FUNCTION_BLOCK SPLIT_AD_INTO_AQ (* this Function splits the 16 AQ (QUARTER) adapters from a AD (DWORD) *)
  (* Standard: 61499-2; Description: Copyright (c) 2026 Meisterschulen am Ostbahnhof SPDX-License-Identifier: EPL-2.0 *)
  (* Version 1.0, 2026-05-16, Franz Höpfinger, Meisterschulen am Ostbahnhof, initial API and implementation and/or initial documentation *)
  PACKAGE adapter::splitting;
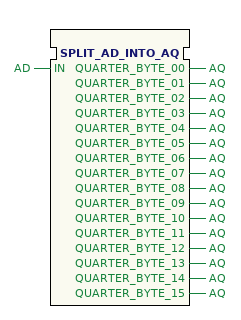
  SOCKETS
    IN : adapter::types::unidirectional::AD; (* DWORD Input *)
  END_SOCKETS
  PLUGS
    QUARTER_BYTE_00 : adapter::types::unidirectional::AQ; (* Quarter 0 *)
    QUARTER_BYTE_01 : adapter::types::unidirectional::AQ; (* Quarter 1 *)
    QUARTER_BYTE_02 : adapter::types::unidirectional::AQ; (* Quarter 2 *)
    QUARTER_BYTE_03 : adapter::types::unidirectional::AQ; (* Quarter 3 *)
    QUARTER_BYTE_04 : adapter::types::unidirectional::AQ; (* Quarter 4 *)
    QUARTER_BYTE_05 : adapter::types::unidirectional::AQ; (* Quarter 5 *)
    QUARTER_BYTE_06 : adapter::types::unidirectional::AQ; (* Quarter 6 *)
    QUARTER_BYTE_07 : adapter::types::unidirectional::AQ; (* Quarter 7 *)
    QUARTER_BYTE_08 : adapter::types::unidirectional::AQ; (* Quarter 8 *)
    QUARTER_BYTE_09 : adapter::types::unidirectional::AQ; (* Quarter 9 *)
    QUARTER_BYTE_10 : adapter::types::unidirectional::AQ; (* Quarter 10 *)
    QUARTER_BYTE_11 : adapter::types::unidirectional::AQ; (* Quarter 11 *)
    QUARTER_BYTE_12 : adapter::types::unidirectional::AQ; (* Quarter 12 *)
    QUARTER_BYTE_13 : adapter::types::unidirectional::AQ; (* Quarter 13 *)
    QUARTER_BYTE_14 : adapter::types::unidirectional::AQ; (* Quarter 14 *)
    QUARTER_BYTE_15 : adapter::types::unidirectional::AQ; (* Quarter 15 *)
  END_PLUGS
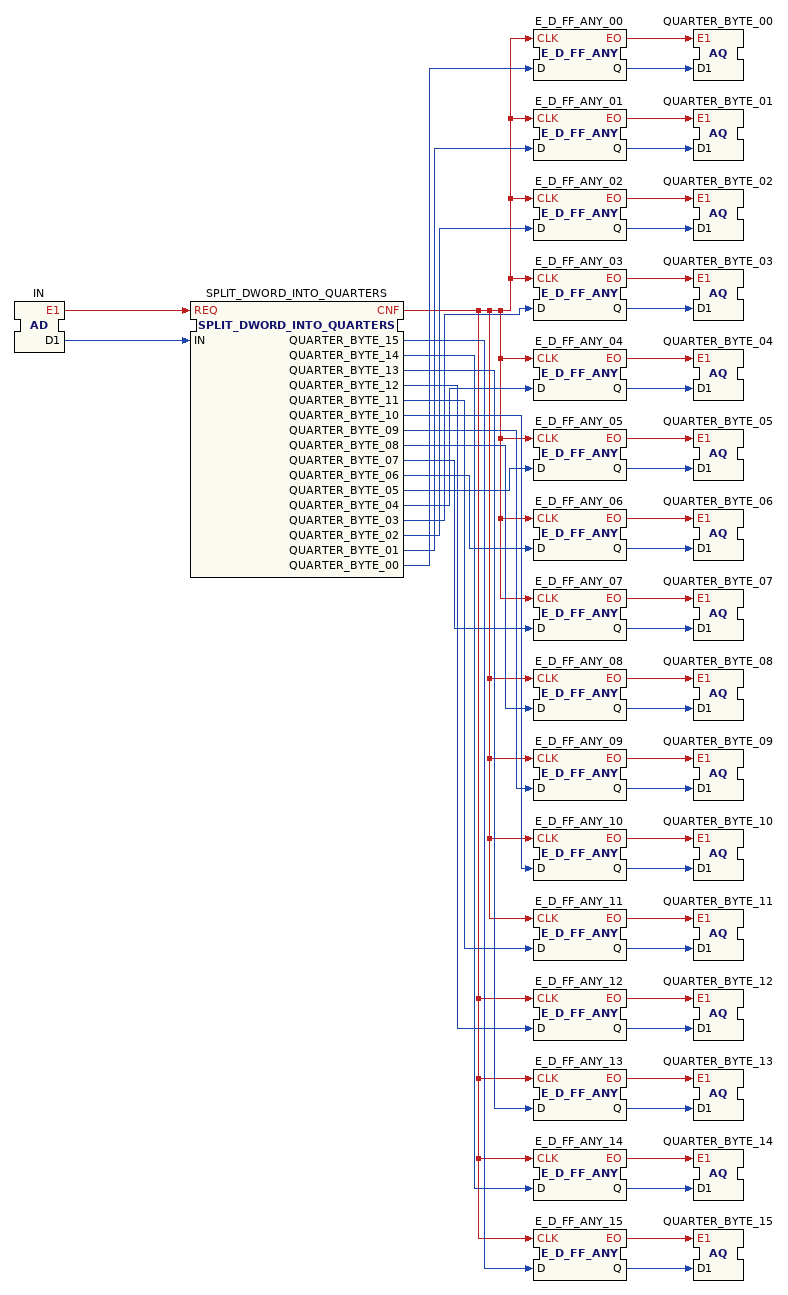
  FBS
    E_D_FF_ANY_00 : iec61499::events::E_D_FF_ANY;
    E_D_FF_ANY_01 : iec61499::events::E_D_FF_ANY;
    E_D_FF_ANY_02 : iec61499::events::E_D_FF_ANY;
    E_D_FF_ANY_03 : iec61499::events::E_D_FF_ANY;
    E_D_FF_ANY_04 : iec61499::events::E_D_FF_ANY;
    E_D_FF_ANY_05 : iec61499::events::E_D_FF_ANY;
    E_D_FF_ANY_06 : iec61499::events::E_D_FF_ANY;
    E_D_FF_ANY_07 : iec61499::events::E_D_FF_ANY;
    E_D_FF_ANY_08 : iec61499::events::E_D_FF_ANY;
    E_D_FF_ANY_09 : iec61499::events::E_D_FF_ANY;
    E_D_FF_ANY_10 : iec61499::events::E_D_FF_ANY;
    E_D_FF_ANY_11 : iec61499::events::E_D_FF_ANY;
    E_D_FF_ANY_12 : iec61499::events::E_D_FF_ANY;
    E_D_FF_ANY_13 : iec61499::events::E_D_FF_ANY;
    E_D_FF_ANY_14 : iec61499::events::E_D_FF_ANY;
    E_D_FF_ANY_15 : iec61499::events::E_D_FF_ANY;
    SPLIT_DWORD_INTO_QUARTERS : eclipse4diac::utils::splitting::SPLIT_DWORD_INTO_QUARTERS;
  END_FBS
  EVENT_CONNECTIONS
    IN.E1 TO SPLIT_DWORD_INTO_QUARTERS.REQ;
    SPLIT_DWORD_INTO_QUARTERS.CNF TO E_D_FF_ANY_00.CLK;
    SPLIT_DWORD_INTO_QUARTERS.CNF TO E_D_FF_ANY_01.CLK;
    SPLIT_DWORD_INTO_QUARTERS.CNF TO E_D_FF_ANY_02.CLK;
    SPLIT_DWORD_INTO_QUARTERS.CNF TO E_D_FF_ANY_03.CLK;
    SPLIT_DWORD_INTO_QUARTERS.CNF TO E_D_FF_ANY_04.CLK;
    SPLIT_DWORD_INTO_QUARTERS.CNF TO E_D_FF_ANY_05.CLK;
    SPLIT_DWORD_INTO_QUARTERS.CNF TO E_D_FF_ANY_06.CLK;
    SPLIT_DWORD_INTO_QUARTERS.CNF TO E_D_FF_ANY_07.CLK;
    SPLIT_DWORD_INTO_QUARTERS.CNF TO E_D_FF_ANY_08.CLK;
    SPLIT_DWORD_INTO_QUARTERS.CNF TO E_D_FF_ANY_09.CLK;
    SPLIT_DWORD_INTO_QUARTERS.CNF TO E_D_FF_ANY_10.CLK;
    SPLIT_DWORD_INTO_QUARTERS.CNF TO E_D_FF_ANY_11.CLK;
    SPLIT_DWORD_INTO_QUARTERS.CNF TO E_D_FF_ANY_12.CLK;
    SPLIT_DWORD_INTO_QUARTERS.CNF TO E_D_FF_ANY_13.CLK;
    SPLIT_DWORD_INTO_QUARTERS.CNF TO E_D_FF_ANY_14.CLK;
    SPLIT_DWORD_INTO_QUARTERS.CNF TO E_D_FF_ANY_15.CLK;
    E_D_FF_ANY_00.EO TO QUARTER_BYTE_00.E1;
    E_D_FF_ANY_01.EO TO QUARTER_BYTE_01.E1;
    E_D_FF_ANY_02.EO TO QUARTER_BYTE_02.E1;
    E_D_FF_ANY_03.EO TO QUARTER_BYTE_03.E1;
    E_D_FF_ANY_04.EO TO QUARTER_BYTE_04.E1;
    E_D_FF_ANY_05.EO TO QUARTER_BYTE_05.E1;
    E_D_FF_ANY_06.EO TO QUARTER_BYTE_06.E1;
    E_D_FF_ANY_07.EO TO QUARTER_BYTE_07.E1;
    E_D_FF_ANY_08.EO TO QUARTER_BYTE_08.E1;
    E_D_FF_ANY_09.EO TO QUARTER_BYTE_09.E1;
    E_D_FF_ANY_10.EO TO QUARTER_BYTE_10.E1;
    E_D_FF_ANY_11.EO TO QUARTER_BYTE_11.E1;
    E_D_FF_ANY_12.EO TO QUARTER_BYTE_12.E1;
    E_D_FF_ANY_13.EO TO QUARTER_BYTE_13.E1;
    E_D_FF_ANY_14.EO TO QUARTER_BYTE_14.E1;
    E_D_FF_ANY_15.EO TO QUARTER_BYTE_15.E1;
  END_CONNECTIONS
  DATA_CONNECTIONS
    IN.D1 TO SPLIT_DWORD_INTO_QUARTERS.IN;
    SPLIT_DWORD_INTO_QUARTERS.QUARTER_BYTE_15 TO E_D_FF_ANY_15.D;
    SPLIT_DWORD_INTO_QUARTERS.QUARTER_BYTE_14 TO E_D_FF_ANY_14.D;
    SPLIT_DWORD_INTO_QUARTERS.QUARTER_BYTE_13 TO E_D_FF_ANY_13.D;
    SPLIT_DWORD_INTO_QUARTERS.QUARTER_BYTE_12 TO E_D_FF_ANY_12.D;
    SPLIT_DWORD_INTO_QUARTERS.QUARTER_BYTE_11 TO E_D_FF_ANY_11.D;
    SPLIT_DWORD_INTO_QUARTERS.QUARTER_BYTE_10 TO E_D_FF_ANY_10.D;
    SPLIT_DWORD_INTO_QUARTERS.QUARTER_BYTE_09 TO E_D_FF_ANY_09.D;
    SPLIT_DWORD_INTO_QUARTERS.QUARTER_BYTE_08 TO E_D_FF_ANY_08.D;
    SPLIT_DWORD_INTO_QUARTERS.QUARTER_BYTE_07 TO E_D_FF_ANY_07.D;
    SPLIT_DWORD_INTO_QUARTERS.QUARTER_BYTE_06 TO E_D_FF_ANY_06.D;
    SPLIT_DWORD_INTO_QUARTERS.QUARTER_BYTE_05 TO E_D_FF_ANY_05.D;
    SPLIT_DWORD_INTO_QUARTERS.QUARTER_BYTE_04 TO E_D_FF_ANY_04.D;
    SPLIT_DWORD_INTO_QUARTERS.QUARTER_BYTE_03 TO E_D_FF_ANY_03.D;
    SPLIT_DWORD_INTO_QUARTERS.QUARTER_BYTE_02 TO E_D_FF_ANY_02.D;
    SPLIT_DWORD_INTO_QUARTERS.QUARTER_BYTE_01 TO E_D_FF_ANY_01.D;
    SPLIT_DWORD_INTO_QUARTERS.QUARTER_BYTE_00 TO E_D_FF_ANY_00.D;
    E_D_FF_ANY_00.Q TO QUARTER_BYTE_00.D1;
    E_D_FF_ANY_01.Q TO QUARTER_BYTE_01.D1;
    E_D_FF_ANY_02.Q TO QUARTER_BYTE_02.D1;
    E_D_FF_ANY_03.Q TO QUARTER_BYTE_03.D1;
    E_D_FF_ANY_04.Q TO QUARTER_BYTE_04.D1;
    E_D_FF_ANY_05.Q TO QUARTER_BYTE_05.D1;
    E_D_FF_ANY_06.Q TO QUARTER_BYTE_06.D1;
    E_D_FF_ANY_07.Q TO QUARTER_BYTE_07.D1;
    E_D_FF_ANY_08.Q TO QUARTER_BYTE_08.D1;
    E_D_FF_ANY_09.Q TO QUARTER_BYTE_09.D1;
    E_D_FF_ANY_10.Q TO QUARTER_BYTE_10.D1;
    E_D_FF_ANY_11.Q TO QUARTER_BYTE_11.D1;
    E_D_FF_ANY_12.Q TO QUARTER_BYTE_12.D1;
    E_D_FF_ANY_13.Q TO QUARTER_BYTE_13.D1;
    E_D_FF_ANY_14.Q TO QUARTER_BYTE_14.D1;
    E_D_FF_ANY_15.Q TO QUARTER_BYTE_15.D1;
  END_CONNECTIONS
END_FUNCTION_BLOCK
